TYPE ST_St040_IO_OUT :
STRUCT
	// outputs OptischeKontrolle	
	nCamPrgAs	: INT;
	nCamPrgBs	: INT;
	
	bLedAs		: BOOL;
	bLedBs		: BOOL;
END_STRUCT
END_TYPE

(* stored: Version 1.1.0.1
   DUT ST_St040_IO_OUT: Id {f3204e21-9c58-402b-b0db-b1fb83143965} *)
